70 : DIST(COND:=COND,MD0=>MD850,MD1=>MD851,MD2=>MD852,MD3=>MD853,MD4=>MD854);
71 : DIST(COND:=COND,MD0=>MD855,MD1=>MD856,MD2=>MD857,MD3=>MD858,MD4=>MD859);
72 : DIST(COND:=COND,MD0=>MD860,MD1=>MD861,MD2=>MD862,MD3=>MD863,MD4=>MD864);
73 : DIST(COND:=COND,MD0=>MD865,MD1=>MD866,MD2=>MD867,MD3=>MD868,MD4=>MD869);
74 : DIST(COND:=COND,MD0=>MD870,MD1=>MD871,MD2=>MD872,MD3=>MD873,MD4=>MD874);
75 : DIST(COND:=COND,MD0=>MD875,MD1=>MD876,MD2=>MD877,MD3=>MD878,MD4=>MD879);
76 : DIST(COND:=COND,MD0=>MD880,MD1=>MD881,MD2=>MD882,MD3=>MD883,MD4=>MD884);
77 : DIST(COND:=COND,MD0=>MD885,MD1=>MD886,MD2=>MD887,MD3=>MD888,MD4=>MD889);
78 : DIST(COND:=COND,MD0=>MD890,MD1=>MD891,MD2=>MD892,MD3=>MD893,MD4=>MD894);
79 : DIST(COND:=COND,MD0=>MD895,MD1=>MD896,MD2=>MD897,MD3=>MD898,MD4=>MD899);

80 : DIST(COND:=COND,MD0=>MD900,MD1=>MD901,MD2=>MD902,MD3=>MD903,MD4=>MD904);
81 : DIST(COND:=COND,MD0=>MD905,MD1=>MD906,MD2=>MD907,MD3=>MD908,MD4=>MD909);
82 : DIST(COND:=COND,MD0=>MD910,MD1=>MD911,MD2=>MD912,MD3=>MD913,MD4=>MD914);
83 : DIST(COND:=COND,MD0=>MD915,MD1=>MD916,MD2=>MD917,MD3=>MD918,MD4=>MD919);
84 : DIST(COND:=COND,MD0=>MD920,MD1=>MD921,MD2=>MD922,MD3=>MD923,MD4=>MD924);
85 : DIST(COND:=COND,MD0=>MD925,MD1=>MD926,MD2=>MD927,MD3=>MD928,MD4=>MD929);
86 : DIST(COND:=COND,MD0=>MD930,MD1=>MD931,MD2=>MD932,MD3=>MD933,MD4=>MD934);
87 : DIST(COND:=COND,MD0=>MD935,MD1=>MD936,MD2=>MD937,MD3=>MD938,MD4=>MD939);
88 : DIST(COND:=COND,MD0=>MD940,MD1=>MD941,MD2=>MD942,MD3=>MD943,MD4=>MD944);
89 : DIST(COND:=COND,MD0=>MD945,MD1=>MD946,MD2=>MD947,MD3=>MD948,MD4=>MD949);

90 : DIST(COND:=COND,MD0=>MD950,MD1=>MD951,MD2=>MD952,MD3=>MD953,MD4=>MD954);
91 : DIST(COND:=COND,MD0=>MD955,MD1=>MD956,MD2=>MD957,MD3=>MD958,MD4=>MD959);
92 : DIST(COND:=COND,MD0=>MD960,MD1=>MD961,MD2=>MD962,MD3=>MD963,MD4=>MD964);
93 : DIST(COND:=COND,MD0=>MD965,MD1=>MD966,MD2=>MD967,MD3=>MD968,MD4=>MD969);
94 : DIST(COND:=COND,MD0=>MD970,MD1=>MD971,MD2=>MD972,MD3=>MD973,MD4=>MD974);
95 : DIST(COND:=COND,MD0=>MD975,MD1=>MD976,MD2=>MD977,MD3=>MD978,MD4=>MD979);
96 : DIST(COND:=COND,MD0=>MD980,MD1=>MD981,MD2=>MD982,MD3=>MD983,MD4=>MD984);
97 : DIST(COND:=COND,MD0=>MD985,MD1=>MD986,MD2=>MD987,MD3=>MD988,MD4=>MD989);
98 : DIST(COND:=COND,MD0=>MD990,MD1=>MD991,MD2=>MD992,MD3=>MD993,MD4=>MD994);
99 : DIST(COND:=COND,MD0=>MD995,MD1=>MD996,MD2=>MD997,MD3=>MD998,MD4=>MD999);

END_CASE;
          
END_FUNCTION_BLOCK

(* Запись элемента в выходные массивы *)
FUNCTION_BLOCK WriteItem
  VAR_INPUT
    PIT : TPos8 := -1;  (* Индекс элемента в массиве ITS *)
  END_VAR
  VAR
    Cond : TCond;  (* Состояние элемента *)
    msg : STRING := '';  (* TEST *)
    _SetCond : SetCond;
  END_VAR

            (* Запись состояния в регистры *)
Cond    := get_cn(PIT);
Cond.ID := it_id(PIT);
(*TEST*)
(* #53 - ID = 16761, 0x4179, REG = 3578-3587 *)
(*
if (Cond.ID = 16761) then 
  msg := MakeMsg(msg, '= TEST1 [', ID2Str(IT_ID(PIT)), ',');
  msg := MakeMsg(msg, SINT_TO_STRING(PIT), ',');
  msg := MakeMsg(msg, 'Tmid=', REAL_TO_STRING(INT_TO_REAL(Cond.Tmid)/100.0), ',');
  msg := MakeMsg(msg, 'Tmax=', REAL_TO_STRING(INT_TO_REAL(Cond.Tmax.v)/100.0), ',');
  msg := MakeMsg(msg,  INT_TO_STRING(Cond.Tmax.i[0]), ',');
  msg := MakeMsg(msg,  INT_TO_STRING(Cond.Tmax.i[1]), ',');
  msg := MakeMsg(msg,  INT_TO_STRING(Cond.Tmax.i[2]), ']');
  msg := LogMsg(msg);
end_if;
*)
_SetCond(I := SINT_TO_UINT(PIT), COND := Cond);
          
END_FUNCTION_BLOCK

(* Вывод результатов в регистры *)
PROGRAM P_RES
  VAR_EXTERNAL
    f_Res : BOOL;  (* Флаг выкладки результатов *)
    HDR : THead;  (* Заголовок модели *)
    ITS : TItems;  (* Массив элементов модели *)
  END_VAR
  VAR
    pit : TPos8 := 0;  (* Позиция элемента *)
    Sh : TShape;  (* Фигура элемента *)
    Pt : TPoint;  (* Точка *)
    Off : P_INT;  (* Offset *)
    PGR : TPos8 := -1;  (* Позиция сетки *)
    I : INT := 0;  (* Индекс сетки X *)
    J : INT := 0;  (* Индекс сетки Y *)
    K : INT := 0;  (* Индекс сетки Z *)
    Dot : TDot;  (* Точка сетки *)
    bRes : BOOL := false;  (* Бинарный результат *)
    iRes : TError := E_SUCCESS;  (* Код ошибки *)
    iLog : INT := 0;  (* Счётчик строк протокола *)
    msg : STRING := '';  (* Сообщение в протокол *)
    _WriteItem : WriteItem;  (* Функция записи элемента *)
    _Grid2ul : Grid2ul;
    _GetHead : GetHead;
  END_VAR

            (* Считывание заголовка *)
_GetHead(HEAD => HDR);

(* Test *)
(* if (HDR.ID = 100)  then HDR.ID := 99; end_if; *)
(*
HDR.ID := 100;
HDR.Ax := 2;
HDR.pX := 1800;
HDR.pY := 620;
HDR.pZ := 1575;
*)
(* =1= Протоколирование на консоль === *)
bRes := Do_LogCond(ID2PIT(0));

(* =2= Запись массива элементов в регистры === *)
(*msg:=LogMsg('Write items ... '); *)
FOR pit := 0 TO HDR.Ni-1 DO 
  _WriteItem(PIT := pit);
  (*
  if (len(msg)=0) then msg := MakeMsg(' - Updated items: '); end_if;
  msg := MakeMsg(msg, ' [', ID2Str(IT_ID(pit)), ',');
  msg := MakeMsg(msg,       SINT_TO_STRING(pit), ']');
  if (mod((pit+1),5)=0) then msg:=LogMsg(MakeMsg(msg, ';')); end_if;
  *)
END_FOR; 
(* if (len(msg)>0) then msg:=LogMsg(MakeMsg(msg, ';')); end_if; *)

(* =3= Вывод T-поля объекта [POS=HDR.ID] в регистры === *)
msg:=LogMsg(MakeMsg(msg, '===== T-Field START ====='));      

pit := UINT_TO_SINT(HDR.ID); (* it_pos(ID2PIT(HDR.ID)); *)
if (pit >= 0 and pit < HDR.Ni) then 

  (* Вывод поля обычного элемента *)
  Sh := get_sh(pit);
  _Grid2ul(HGR := its_gr(0), PGR := pit, SH := Sh, iRes=>iRes);
  
elsif (pit = 100) then (* Вывод поля поверхности *)
  
  Sh := _surf(
    ID2PIT(0), 
    UINT_TO_USINT(HDR.Ax), 
    INT_TO_REAL(HDR.pX), 
    INT_TO_REAL(HDR.pY), 
    INT_TO_REAL(HDR.pZ)
  );
  (*Sh := get_sh(0);*)
  ITS.Sh[pit] := Sh;
  
  (* Линковка узлов *)
  iLog := 0;
  for I:=0 to Sh.Kn[0]-1 do
    for J:=0 to Sh.Kn[1]-1 do
      for K:=0 to Sh.Kn[2]-1 do
      
        Dot := link_var(its_gr2(0), 0, Sh, I, J, K);
        (*
        Pt  := Sh_Dot2Point(Sh, I, J, K);
        Dot := Do_FindDot(Pt[0], Pt[1], Pt[2]);
        Off := knoff(Sh.Kn[0], Sh.Kn[1], Sh.Kn[2], I,J,K);
        PGR := set_var( its_gr2(0), 0, Off, _ref(int_to_sint(Dot.v), Dot));
        *)
        
        (*
        if (false or iLog<80) then  
          if (len(msg)=0) then msg := MakeMsg(' =!=> '); end_if;
          msg := MakeMsg(msg, '[', INT_TO_STRING(REAL_TO_INT(Pt[0])), ',');
          msg := MakeMsg(msg,  '', INT_TO_STRING(REAL_TO_INT(Pt[1])), ',');
          msg := MakeMsg(msg,  '', INT_TO_STRING(REAL_TO_INT(Pt[2])), ']');
          if (mod((iLog+1),8)=0) then msg:=LogMsg(MakeMsg(msg, ';')); end_if;
          iLog:=iLog+1;
        end_if;
        *)
        (*
        if (iLog<80) then  
          if (len(msg)=0) then msg := MakeMsg(' =!=> '); end_if;
          msg := MakeMsg(msg, '[', INT_TO_STRING(Dot.v), ',');
          msg := MakeMsg(msg,  '', INT_TO_STRING(Dot.a[0]), ',');
          msg := MakeMsg(msg,  '', INT_TO_STRING(Dot.a[1]), ',');
          msg := MakeMsg(msg,  '', INT_TO_STRING(Dot.a[2]), ']');
          if (mod((iLog+1),8)=0) then msg:=LogMsg(MakeMsg(msg, ';')); end_if;
          iLog:=iLog+1;
        end_if;
        *)
      end_for;
    end_for;
  end_for;
  if (len(msg)>0) then msg:=LogMsg(MakeMsg(msg, ';')); end_if;
  
  _Grid2ul(HGR := its_gr2(0), PGR := 0, SH := Sh, iRes=>iRes);
  
else (* ошибка позиции *)
  {}

end_if;
msg:=LogMsg(MakeMsg(msg, '===== T-Field (END) ====='));      

(* Сброс флага *)
f_Res := FALSE;

          
END_PROGRAM

FUNCTION UDI2REAL : REAL
  VAR_INPUT
    VALUE : UDINT := 0;
  END_VAR
  VAR
    tmp : REAL := 0.0;
  END_VAR

            {{
  union { UDINT  udint; float real; } value;
  value.udint = VALUE;
  TMP = value.real;
}}
UDI2REAL := TMP;

          
END_FUNCTION

(* Компоновка материала *)
FUNCTION m_mat : TMat
  VAR_INPUT
    MD0 : UDINT;
    MD1 : UDINT;
    MD2 : UDINT;
    MD3 : UDINT;
  END_VAR

            m_mat.KT := UDI2REAL(MD0);
m_mat.CP := UDI2REAL(MD1);
m_mat.PL := UDI2REAL(MD2);
m_mat.MD := UDI2REAL(MD3);

          
END_FUNCTION

(* Чтение материала из регистров *)
FUNCTION_BLOCK GetMat
  VAR_EXTERNAL
    MD22 : UDINT;
    MD23 : UDINT;
    MD24 : UDINT;
    MD25 : UDINT;
    MD26 : UDINT;
    MD27 : UDINT;
    MD28 : UDINT;
    MD29 : UDINT;
    MD30 : UDINT;
    MD31 : UDINT;
    MD32 : UDINT;
    MD33 : UDINT;
    MD34 : UDINT;
    MD35 : UDINT;
    MD36 : UDINT;
    MD37 : UDINT;
    MD38 : UDINT;
    MD39 : UDINT;
    MD40 : UDINT;
    MD41 : UDINT;
    MD42 : UDINT;
    MD43 : UDINT;
    MD44 : UDINT;
    MD45 : UDINT;
    MD46 : UDINT;
    MD47 : UDINT;
    MD48 : UDINT;
    MD49 : UDINT;
    MD50 : UDINT;
    MD51 : UDINT;
    MD52 : UDINT;
    MD53 : UDINT;
    MD54 : UDINT;
    MD55 : UDINT;
    MD56 : UDINT;
    MD57 : UDINT;
    MD58 : UDINT;
    MD59 : UDINT;
    MD60 : UDINT;
    MD61 : UDINT;
    MD62 : UDINT;
    MD63 : UDINT;
    MD64 : UDINT;
    MD65 : UDINT;
    MD66 : UDINT;
    MD67 : UDINT;
    MD68 : UDINT;
    MD69 : UDINT;
  END_VAR
  VAR_INPUT
    I : SINT := 0;  (* Индекс материала *)
  END_VAR
  VAR_OUTPUT
    MAT : TMat;  (* Объект "материал" *)
  END_VAR

            CASE i OF
0 : MAT := m_mat(MD22,MD23,MD24,MD25);
1 : MAT := m_mat(MD26,MD27,MD28,MD29);
2 : MAT := m_mat(MD30,MD31,MD32,MD33);
3 : MAT := m_mat(MD34,MD35,MD36,MD37);
4 : MAT := m_mat(MD38,MD39,MD40,MD41);
5 : MAT := m_mat(MD42,MD43,MD44,MD45);
6 : MAT := m_mat(MD46,MD47,MD48,MD49);
7 : MAT := m_mat(MD50,MD51,MD52,MD53);
8 : MAT := m_mat(MD54,MD55,MD56,MD57);
9 : MAT := m_mat(MD58,MD59,MD60,MD61);
10: MAT := m_mat(MD62,MD63,MD64,MD65);
11: MAT := m_mat(MD66,MD67,MD68,MD69);
END_CASE;
          
END_FUNCTION_BLOCK

(* Компоновка профиля *)
FUNCTION m_prof : TProf
  VAR_INPUT
    MD0 : UDINT;
    MD1 : UDINT;
    MD2 : UDINT;
    MD3 : UDINT;
    MD4 : UDINT;
    MD5 : UDINT;
  END_VAR

            m_prof[0].A := UINT_TO_SINT(UDINT_TO_UINT(MD0/65536)/256);
m_prof[0].B := UINT_TO_SINT(mod(UDINT_TO_UINT(MD0/65536),256));
m_prof[1].A := UINT_TO_SINT(UDINT_TO_UINT(mod(MD0,65536))/256);
m_prof[1].B := UINT_TO_SINT(mod(UDINT_TO_UINT(mod(MD0,65536)),256));

m_prof[2].A := UINT_TO_SINT(UDINT_TO_UINT(MD1/65536)/256);
m_prof[2].B := UINT_TO_SINT(mod(UDINT_TO_UINT(MD1/65536),256));
m_prof[3].A := UINT_TO_SINT(UDINT_TO_UINT(mod(MD1,65536))/256);
m_prof[3].B := UINT_TO_SINT(mod(UDINT_TO_UINT(mod(MD1,65536)),256));

m_prof[4].A := UINT_TO_SINT(UDINT_TO_UINT(MD2/65536)/256);
m_prof[4].B := UINT_TO_SINT(mod(UDINT_TO_UINT(MD2/65536),256));
m_prof[5].A := UINT_TO_SINT(UDINT_TO_UINT(mod(MD2,65536))/256);
m_prof[5].B := UINT_TO_SINT(mod(UDINT_TO_UINT(mod(MD2,65536)),256));

m_prof[6].A := UINT_TO_SINT(UDINT_TO_UINT(MD3/65536)/256);
m_prof[6].B := UINT_TO_SINT(mod(UDINT_TO_UINT(MD3/65536),256));
m_prof[7].A := UINT_TO_SINT(UDINT_TO_UINT(mod(MD3,65536))/256);
m_prof[7].B := UINT_TO_SINT(mod(UDINT_TO_UINT(mod(MD3,65536)),256));

m_prof[8].A := UINT_TO_SINT(UDINT_TO_UINT(MD4/65536)/256);
m_prof[8].B := UINT_TO_SINT(mod(UDINT_TO_UINT(MD4/65536),256));
m_prof[9].A := UINT_TO_SINT(UDINT_TO_UINT(mod(MD4,65536))/256);
m_prof[9].B := UINT_TO_SINT(mod(UDINT_TO_UINT(mod(MD4,65536)),256));

m_prof[10].A := UINT_TO_SINT(UDINT_TO_UINT(MD5/65536)/256);
m_prof[10].B := UINT_TO_SINT(mod(UDINT_TO_UINT(MD5/65536),256));
m_prof[11].A := UINT_TO_SINT(UDINT_TO_UINT(mod(MD5,65536))/256);
m_prof[11].B := UINT_TO_SINT(mod(UDINT_TO_UINT(mod(MD5,65536)),256));

          
END_FUNCTION

(* Чтение профиля из регистров *)
FUNCTION_BLOCK GetProf
  VAR_EXTERNAL
    MD120 : UDINT;
    MD121 : UDINT;
    MD122 : UDINT;
    MD123 : UDINT;
    MD124 : UDINT;
    MD125 : UDINT;
    MD126 : UDINT;
    MD127 : UDINT;
    MD128 : UDINT;
    MD129 : UDINT;
    MD130 : UDINT;
    MD131 : UDINT;
    MD132 : UDINT;
    MD133 : UDINT;
    MD134 : UDINT;
    MD135 : UDINT;
    MD136 : UDINT;
    MD137 : UDINT;
    MD138 : UDINT;
    MD139 : UDINT;
    MD140 : UDINT;
    MD141 : UDINT;
    MD142 : UDINT;
    MD143 : UDINT;
    MD144 : UDINT;
    MD145 : UDINT;
    MD146 : UDINT;
    MD147 : UDINT;
    MD148 : UDINT;
    MD149 : UDINT;
    MD150 : UDINT;
    MD151 : UDINT;
    MD152 : UDINT;
    MD153 : UDINT;
    MD154 : UDINT;
    MD155 : UDINT;
    MD156 : UDINT;
    MD157 : UDINT;
    MD158 : UDINT;
    MD159 : UDINT;
    MD160 : UDINT;
    MD161 : UDINT;
    MD162 : UDINT;
    MD163 : UDINT;
    MD164 : UDINT;
    MD165 : UDINT;
    MD166 : UDINT;
    MD167 : UDINT;
    MD168 : UDINT;
    MD169 : UDINT;
    MD170 : UDINT;
    MD171 : UDINT;
    MD172 : UDINT;
    MD173 : UDINT;
    MD174 : UDINT;
    MD175 : UDINT;
    MD176 : UDINT;
    MD177 : UDINT;
    MD178 : UDINT;
    MD179 : UDINT;
    MD180 : UDINT;
    MD181 : UDINT;
    MD182 : UDINT;
    MD183 : UDINT;
    MD184 : UDINT;
    MD185 : UDINT;
    MD186 : UDINT;
    MD187 : UDINT;
    MD188 : UDINT;
    MD189 : UDINT;
    MD190 : UDINT;
    MD191 : UDINT;
    MD192 : UDINT;
    MD193 : UDINT;
    MD194 : UDINT;
    MD195 : UDINT;
    MD196 : UDINT;
    MD197 : UDINT;
    MD198 : UDINT;
    MD199 : UDINT;
    MD200 : UDINT;
    MD201 : UDINT;
    MD202 : UDINT;
    MD203 : UDINT;
    MD204 : UDINT;
    MD205 : UDINT;
    MD206 : UDINT;
    MD207 : UDINT;
    MD208 : UDINT;
    MD209 : UDINT;
    MD210 : UDINT;
    MD211 : UDINT;
    MD212 : UDINT;
    MD213 : UDINT;
    MD214 : UDINT;
    MD215 : UDINT;
    MD216 : UDINT;
    MD217 : UDINT;
    MD218 : UDINT;
    MD219 : UDINT;
    MD220 : UDINT;
    MD221 : UDINT;
    MD222 : UDINT;
    MD223 : UDINT;
    MD224 : UDINT;
    MD225 : UDINT;
    MD226 : UDINT;
    MD227 : UDINT;
    MD228 : UDINT;
    MD229 : UDINT;
    MD230 : UDINT;
    MD231 : UDINT;
    MD232 : UDINT;
    MD233 : UDINT;
    MD234 : UDINT;
    MD235 : UDINT;
    MD236 : UDINT;
    MD237 : UDINT;
    MD238 : UDINT;
    MD239 : UDINT;
    MD240 : UDINT;
    MD241 : UDINT;
    MD242 : UDINT;
    MD243 : UDINT;
    MD244 : UDINT;
    MD245 : UDINT;
    MD246 : UDINT;
    MD247 : UDINT;
    MD248 : UDINT;
    MD249 : UDINT;
    MD250 : UDINT;
    MD251 : UDINT;
    MD252 : UDINT;
    MD253 : UDINT;
    MD254 : UDINT;
    MD255 : UDINT;
    MD256 : UDINT;
    MD257 : UDINT;
    MD258 : UDINT;
    MD259 : UDINT;
    MD260 : UDINT;
    MD261 : UDINT;
    MD262 : UDINT;
    MD263 : UDINT;
    MD264 : UDINT;
    MD265 : UDINT;
    MD266 : UDINT;
    MD267 : UDINT;
    MD268 : UDINT;
    MD269 : UDINT;
    MD270 : UDINT;
    MD271 : UDINT;
    MD272 : UDINT;
    MD273 : UDINT;
    MD274 : UDINT;
    MD275 : UDINT;
    MD276 : UDINT;
    MD277 : UDINT;
    MD278 : UDINT;
    MD279 : UDINT;
    MD280 : UDINT;
    MD281 : UDINT;
    MD282 : UDINT;
    MD283 : UDINT;
    MD284 : UDINT;
    MD285 : UDINT;
    MD286 : UDINT;
    MD287 : UDINT;
    MD288 : UDINT;
    MD289 : UDINT;
    MD290 : UDINT;
    MD291 : UDINT;
    MD292 : UDINT;
    MD293 : UDINT;
    MD294 : UDINT;
    MD295 : UDINT;
    MD296 : UDINT;
    MD297 : UDINT;
    MD298 : UDINT;
    MD299 : UDINT;
  END_VAR
  VAR_INPUT
    I : SINT := 0;  (* Индекс профиля *)
  END_VAR
  VAR_OUTPUT
    PROF : TProf;  (* Объект "профиль" *)
  END_VAR

            CASE i OF
0 : PROF := m_prof(MD120,MD121,MD122,MD123,MD124,MD125);
1 : PROF := m_prof(MD126,MD127,MD128,MD129,MD130,MD131);
2 : PROF := m_prof(MD132,MD133,MD134,MD135,MD136,MD137);
3 : PROF := m_prof(MD138,MD139,MD140,MD141,MD142,MD143);
4 : PROF := m_prof(MD144,MD145,MD146,MD147,MD148,MD149);
5 : PROF := m_prof(MD150,MD151,MD152,MD153,MD154,MD155);
6 : PROF := m_prof(MD156,MD157,MD158,MD159,MD160,MD161);
7 : PROF := m_prof(MD162,MD163,MD164,MD165,MD166,MD167);
8 : PROF := m_prof(MD168,MD169,MD170,MD171,MD172,MD173);
9 : PROF := m_prof(MD174,MD175,MD176,MD177,MD178,MD179);
10: PROF := m_prof(MD180,MD181,MD182,MD183,MD184,MD185);
11: PROF := m_prof(MD186,MD187,MD188,MD189,MD190,MD191);
12: PROF := m_prof(MD192,MD193,MD194,MD195,MD196,MD197);
13: PROF := m_prof(MD198,MD199,MD200,MD201,MD202,MD203);
14: PROF := m_prof(MD204,MD205,MD206,MD207,MD208,MD209);
15: PROF := m_prof(MD210,MD211,MD212,MD213,MD214,MD215);
16: PROF := m_prof(MD216,MD217,MD218,MD219,MD220,MD221);
17: PROF := m_prof(MD222,MD223,MD224,MD225,MD226,MD227);
18: PROF := m_prof(MD228,MD229,MD230,MD231,MD232,MD233);
19: PROF := m_prof(MD234,MD235,MD236,MD237,MD238,MD239);
20: PROF := m_prof(MD240,MD241,MD242,MD243,MD244,MD245);
21: PROF := m_prof(MD246,MD247,MD248,MD249,MD250,MD251);
22: PROF := m_prof(MD252,MD253,MD254,MD255,MD256,MD257);
23: PROF := m_prof(MD258,MD259,MD260,MD261,MD262,MD263);
24: PROF := m_prof(MD264,MD265,MD266,MD267,MD268,MD269);
25: PROF := m_prof(MD270,MD271,MD272,MD273,MD274,MD275);
26: PROF := m_prof(MD276,MD277,MD278,MD279,MD280,MD281);
27: PROF := m_prof(MD282,MD283,MD284,MD285,MD286,MD287);
28: PROF := m_prof(MD288,MD289,MD290,MD291,MD292,MD293);
29: PROF := m_prof(MD294,MD295,MD296,MD297,MD298,MD299);
END_CASE;
          
END_FUNCTION_BLOCK

(* Компоновка величины *)
FUNCTION m_val : TVal
  VAR_INPUT
    MD0 : UDINT;
    MD1 : UDINT;
  END_VAR

            m_val.Iv      := UDINT_TO_INT(MD0/65536);
m_val.Vi[0].A := UINT_TO_SINT(UDINT_TO_UINT(mod(MD0,65536))/256);
m_val.Vi[0].B := UINT_TO_SINT(mod(UDINT_TO_UINT(mod(MD0,65536)),256));
m_val.Vi[1].A := UINT_TO_SINT(UDINT_TO_UINT(MD1/65536)/256);
m_val.Vi[1].B := UINT_TO_SINT(mod(UDINT_TO_UINT(MD1/65536),256));
m_val.Vi[2].A := UINT_TO_SINT(UDINT_TO_UINT(mod(MD1,65536))/256);
m_val.Vi[2].B := UINT_TO_SINT(mod(UDINT_TO_UINT(mod(MD1,65536)),256));



          
END_FUNCTION

(* Чтение величины из регистров *)
FUNCTION_BLOCK GetVal
  VAR_EXTERNAL
    MD70 : UDINT;
    MD71 : UDINT;
    MD72 : UDINT;
    MD73 : UDINT;
    MD74 : UDINT;
    MD75 : UDINT;
    MD76 : UDINT;
    MD77 : UDINT;
    MD78 : UDINT;
    MD79 : UDINT;
    MD80 : UDINT;
    MD81 : UDINT;
    MD82 : UDINT;
    MD83 : UDINT;
    MD84 : UDINT;
    MD85 : UDINT;
    MD86 : UDINT;
    MD87 : UDINT;
    MD88 : UDINT;
    MD89 : UDINT;
    MD90 : UDINT;
    MD91 : UDINT;
    MD92 : UDINT;
    MD93 : UDINT;
    MD94 : UDINT;
    MD95 : UDINT;
    MD96 : UDINT;
    MD97 : UDINT;
    MD98 : UDINT;
    MD99 : UDINT;
    MD100 : UDINT;
    MD101 : UDINT;
    MD102 : UDINT;
    MD103 : UDINT;
    MD104 : UDINT;
    MD105 : UDINT;
    MD106 : UDINT;
    MD107 : UDINT;
    MD108 : UDINT;
    MD109 : UDINT;
    MD110 : UDINT;
    MD111 : UDINT;
    MD112 : UDINT;
    MD113 : UDINT;
    MD114 : UDINT;
    MD115 : UDINT;
    MD116 : UDINT;
    MD117 : UDINT;
    MD118 : UDINT;
    MD119 : UDINT;
  END_VAR
  VAR_INPUT
    I : SINT := 0;  (* Индекс величины *)
  END_VAR
  VAR_OUTPUT
    VAL : TVal;  (* Объект "величина" *)
  END_VAR

            CASE i OF
0 : VAL := m_val(MD70,MD71);
1 : VAL := m_val(MD72,MD73);
2 : VAL := m_val(MD74,MD75);
3 : VAL := m_val(MD76,MD77);
4 : VAL := m_val(MD78,MD79);
5 : VAL := m_val(MD80,MD81);
6 : VAL := m_val(MD82,MD83);
7 : VAL := m_val(MD84,MD85);
8 : VAL := m_val(MD86,MD87);
9 : VAL := m_val(MD88,MD89);
10: VAL := m_val(MD90,MD91);
11: VAL := m_val(MD92,MD93);
12: VAL := m_val(MD94,MD95);
13: VAL := m_val(MD96,MD97);
14: VAL := m_val(MD98,MD99);
15: VAL := m_val(MD100,MD101);
16: VAL := m_val(MD102,MD103);
17: VAL := m_val(MD104,MD105);
18: VAL := m_val(MD106,MD107);
19: VAL := m_val(MD108,MD109);
20: VAL := m_val(MD110,MD111);
21: VAL := m_val(MD112,MD113);
22: VAL := m_val(MD114,MD115);
23: VAL := m_val(MD116,MD117);
24: VAL := m_val(MD118,MD119);
END_CASE;
          
END_FUNCTION_BLOCK

(* Алгоритм "Быстрая сортировка" *)
FUNCTION_BLOCK Sort_IDS
  VAR_EXTERNAL
    ITS : TItems;  (* Массив элементов *)
  END_VAR
  VAR_INPUT
    iBegin : TPos8 := 0;  (* Индекс начала сортировки *)
    iEnd : TPos8 := 0;  (* Индекс завершения сортировки *)
  END_VAR
  VAR_OUTPUT
    iRes : TError := E_SUCCESS;  (* Результат выполнения *)
  END_VAR
  VAR
    iL : TPos8;  (* Левая граница *)
    iR : TPos8;  (* Правая граница *)
    LL : TPos8;  (* Левый индекс *)
    RR : TPos8;  (* Правый индекс *)
    Z : P_IDPIT;  (* Средний элемент для сравнения *)
    iS : TPos8;  (* Индекс стека *)
    Stack : ARRAY[0..49] OF TPos8;  (* Стек индексов элементов *)
    fBreak : BOOL;  (* Флаг завершения внешнего цикла *)
    tmp : P_IDPIT;  (* Буфер обмена значениями *)
  END_VAR

            (* Начальные значения *)
iRes  := E_SUCCESS;				
iS    := 0; 
iL    := iBegin; 
iR    := iEnd; 

fBreak := false;
WHILE NOT fBreak DO         (* внешний цикл = "рекурсия" *)
  
	IF iL < iR THEN
    (* Значение среднего элемента в качестве опорного значения *)
		Z := ITS.Pr[WORD_TO_SINT(SHR(UINT_TO_WORD(SINT_TO_UINT(iR)+SINT_TO_UINT(iL)),1))]; 
    
		LL := iL; RR := iR;
		WHILE (LL <= RR) DO     (* внутренний цикл = выделение частей *)
 			(* Сравнение - возрастающий порядок *)
      while (ITS.Pr[LL].A < Z.A) do LL:=LL+1; end_while;
      while (ITS.Pr[RR].A > Z.A) do RR:=RR-1; end_while;
			if LL <= RR then  
        if (LL <> RR) then  (* Обмен значений *)
          tmp := ITS.Pr[RR]; 
          ITS.Pr[RR] := ITS.Pr[LL]; 
          ITS.Pr[LL] := tmp; 
        end_if;        
        LL:=LL+1; RR:=RR-1;
			end_if;
		END_WHILE;

		(* Вставка в стек *)
		IF iS < 49 THEN 
      Stack[iS] := iR;		  (* Отложенная сортировка правой части  *)
      iS := iS+1; 
    ELSE                    (* Стек выбран - ошибка величины стека *)
      fBreak := TRUE; 
      iRes := E_STACKSIZE; 
    END_IF;
      
		iR := MAX(iL, LL-1);    (* Сортировка левой части - в следующем цикле *)
    
  ELSE
    
		IF iS > 0 THEN          (* Теперь сортируем правую часть *)
			iL := iR+1;
			(* Выборка из стека *)
			iS := iS-1;	
			iR:= Stack[iS];
		ELSE                    (* Стек выбран - конец работы *)
      fBreak := TRUE;
		END_IF;
    
	END_IF;
  
END_WHILE; (* Сортировка завершена *)

          
END_FUNCTION_BLOCK

(* Чтение конфигурации из регистров *)
PROGRAM P_CONF
  VAR_EXTERNAL
    STAT : TStat;  (* Состояние выполнения *)
    f_Conf : BOOL;  (* Флаг конфигурирования *)
    HDR : THead;  (* Заголовок модели *)
    STS : TSets;  (* Массив конфигураций *)
    ITS : TItems;  (* Массив элементов *)
  END_VAR
  VAR
    msg : STRING;  (* Строка сообщения *)
    _GetHead : GetHead;  (* ФБ чтения заголовка *)
    _GetMat : GetMat;  (* ФБ чтения материалов *)
    _GetVal : GetVal;  (* ФБ чтения связанных величин *)
    _GetProf : GetProf;  (* ФБ чтения профилей *)
    _ReadItem : ReadItem;  (* ФБ чтения элементов *)
    _Sort_IDS : Sort_IDS;  (* ФБ "быстрая сортировка" *)
    _Process_X : Process_XYZ;
  END_VAR

            (* Локальные переменные *)
VAR
  i,j,k,l : SINT;      (* Индексы в массивах              *)
  iLev    : SINT;      (* Уровень элемента                *)
  pit,idx : TPos8;     (* Индексы элементов               *)
  iPar    : TPos8;     (* Индекс родителя                 *)
  iPrev   : TPos8;     (* Индекс предыдущего элемента     *)
  nRes    : TError;    (* Код результата выполнения       *)
  iRes    : INT;       (* Возвращаемое значение           *)
  it      : TITER;     (* Итератор для обхода дерева      *)
  btRes   : BYTE;      (* Результат проверки точки модели *)
  bRes    : BOOL;
  rRes    : REAL;
  ii      : DINT;
  sibt    : P_SIBT;
END_VAR

(* Установка начальных значений *)
{{
  // Инициализация фиктивного элемента
  //TITEM *pItem0 = __GET_GLOBAL_DUMMY();
  //memset(pItem0,0x00,sizeof(TITEM));
  //pItem0->ID = 0xffff;
  
  // Инициализация состояния ресурса
  TSTAT *pStat = __GET_GLOBAL_STAT();
  *pStat = (TSTAT) {FALSE, TRUE, TERROR__E_SUCCESS, 0, __INIT_STRING};
}}

nRes := E_SUCCESS;          (* Установка кода результата    *)
bRes := st_set_debug(TRUE); (* Установка флага отладки      *) 

msg  := LogMsg('== CONFIG ...');

(* === Чтение и валидация заголовка === *)
_GetHead(HEAD => HDR);

msg := MakeMsg(' - Read header ... (');
msg := MakeMsg(msg, SINT_TO_STRING(HDR.Ni), ', ');
msg := MakeMsg(msg, SINT_TO_STRING(HDR.Nm), ', ');
msg := MakeMsg(msg, SINT_TO_STRING(HDR.Nv), ', ');
msg := MakeMsg(msg, SINT_TO_STRING(HDR.Np), ')');

(* Валидация заголовка *)
if (HDR.Ni= 0 or HDR.Ni>100) then nRes:=E_HEAD; {goto __exit} end_if;
if (HDR.Nm= 0 or HDR.Nm>12)  then nRes:=E_HEAD; {goto __exit} end_if;
if (HDR.Nv< 0 or HDR.Nv>25)  then nRes:=E_HEAD; {goto __exit} end_if;
if (HDR.Np< 0 or HDR.Np>30)  then nRes:=E_HEAD; {goto __exit} end_if;
msg:=LogMsg(MakeMsg(msg, ';'));

(* Проверка периодов расчёта элемента *)
if (HDR.TR[0] = T#0s) then HDR.TR[0]:=T#15s; end_if;
if (HDR.TR[1] = T#0s) then HDR.TR[1]:=T#30s; end_if;
if (HDR.TR[2] = T#0s) then HDR.TR[2]:=T#45s; end_if;
if (HDR.TR[3] = T#0s) then HDR.TR[3]:=T#60s; end_if;

(* === Чтение и валидация массива материалов === *)
msg:=LogMsg('Read materials ... ');
FOR i := 0 TO HDR.Nm-1 DO 
  _GetMat(I:=i, MAT => STS.Mt[i]);
  msg := MakeMsg(' - Get material [', SINT_TO_STRING(i), '] ... (');
  msg := MakeMsg(msg, REAL_TO_STRING(STS.Mt[i].KT), ', ');
  msg := MakeMsg(msg, REAL_TO_STRING(STS.Mt[i].CP), ', ');
  msg := MakeMsg(msg, REAL_TO_STRING(STS.Mt[i].PL), ', ');
  msg := MakeMsg(msg, REAL_TO_STRING(STS.Mt[i].MD), ')');
  (* Валидация *)
  if (STS.Mt[i].KT < 1.0E-8) then nRes:=E_MATER; {goto __exit} end_if;
  if (STS.Mt[i].CP < 1.0E-8) then nRes:=E_MATER; {goto __exit} end_if;
  if (STS.Mt[i].PL < 1.0E-8) then nRes:=E_MATER; {goto __exit} end_if;
  msg:=LogMsg(MakeMsg(msg, ';'));
END_FOR;

(* === Чтение и валидация профилей === *)
msg:=LogMsg('Read profiles ... ');
FOR i := 0 TO HDR.Np-1 DO 
  _GetProf(I:=i, PROF => STS.Pr[i]);
  msg := MakeMsg(' - Get profile [', SINT_TO_STRING(i), '] ...');
  FOR j := 0 TO 11 DO
    msg := MakeMsg(msg, ' (', SINT_TO_STRING(STS.Pr[i][j].A), ',');
    msg := MakeMsg(msg,       SINT_TO_STRING(STS.Pr[i][j].B), ')');
    (* Валидация *)
    if (STS.Pr[i][j].A <    0 or STS.Pr[i][j].A > 100) then nRes:=E_PROFILE; {goto __exit} end_if;
    if (STS.Pr[i][j].B < -100 or STS.Pr[i][j].B > 100) then nRes:=E_PROFILE; {goto __exit} end_if;
  END_FOR;
  msg:=LogMsg(MakeMsg(msg, ';'));
END_FOR;

(* === Чтение и валидация связанных величин === *)
msg:=LogMsg('Read values ... ');
FOR i := 0 TO HDR.Nv-1 DO 
  _GetVal(I:=i, VAL => STS.Vl[i]);
  msg := MakeMsg(' - Get value [', SINT_TO_STRING(i), '] ...');
  if (STS.Vl[i].Iv >=USINT_TO_INT(30) and STS.Vl[i].Iv <> -1) then nRes:=E_VALUE; {goto __exit} end_if;
  FOR j := 0 TO 2 DO
    msg := MakeMsg(msg, ' (', SINT_TO_STRING(STS.Vl[i].Vi[j].A), ',');
    msg := MakeMsg(msg,       SINT_TO_STRING(STS.Vl[i].Vi[j].B), ')');
    (* Валидация *)
    if (STS.Vl[i].Vi[j].A < 0 or STS.Vl[i].Vi[j].A >     100) then nRes:=E_VALUE; {goto __exit} end_if;
    if (STS.Vl[i].Vi[j].B < 0 or STS.Vl[i].Vi[j].B >= HDR.Np) then nRes:=E_VALUE; {goto __exit} end_if;
  END_FOR;
  msg:=LogMsg(MakeMsg(msg, ';'));
END_FOR;

(* === Чтение массива элементов === *)
msg:=LogMsg('Read items ... '); 
FOR pit := 0 TO HDR.Ni-1 DO 
  _ReadItem(PIT := pit, iRes => nRes); 
  
  (* Протоколирование *)
  if (len(msg)=0) then msg := MakeMsg(' - Updated items: '); end_if;
  msg := MakeMsg(msg, ' [', ID2Str(IT_ID(pit)), ',');
  msg := MakeMsg(msg,       SINT_TO_STRING(pit), ']');
  if (mod((pit+1),5)=0) then msg:=LogMsg(MakeMsg(msg, ';')); end_if;
  if (nRes <> E_SUCCESS) then {goto __exit} end_if;
  
  (* Регистрация элемента в массиве IDs (UI->SI)*)
  ITS.Pr[pit].A := ITS.It[pit].ID; 
  ITS.Pr[pit].B := (pit);
END_FOR; 
if (len(msg)>0) then msg:=LogMsg(MakeMsg(msg, ';')); end_if;

(* === Упорядочивание массива по IDs === *)
msg:=LogMsg(MakeMsg('Sort items ... '));
_Sort_IDS(iBegin:=0, iEnd:=HDR.Ni-1, iRes => nRes); 
if (nRes <> E_SUCCESS) then {goto __exit} end_if;

(* === Формирование иерархической структуры === *)
if (ITS.Pr[0].A<>0) then 
  nRes  := E_ROOT; 
  {goto __exit} 
end_if;

(* ROOT settings *)
iPrev := ITS.Pr[0].B;   
iPar  := iPrev;
iLev  := -1;
ITS.It[iPar].Par := -1; 

(* Построение дерева *)
FOR idx := 1 TO HDR.Ni-1 DO
  pit := ITS.Pr[idx].B;   (* Индекс элемента  *)
  l := IT_Lev(pit);       (* Уровень элемента *)
  if (l < 0) then nRes:=E_STRUCT; {goto __exit} end_if;

  (* Определяем индекс родителя iPar *)  
  if (l <> iLev) then     (* Смена уровня вложенности - смена родителя *)
    (* Нахождение родителя для текущего элемента *)
    if (l > iLev) then    (* Спускаемся на уровень вниз  *)
      (* Возможен спуск только на одну ступень (!) *)
      if (l-iLev <> 1) then nRes:=E_STRUCT; {goto __exit} end_if;
      (* Предыдущий элемент должен быть родительским *)
      (*if (not ITS.IT[iPrev].bP) then nRes:=E_STRUCT; {goto __exit} end_if;*)
      iPar := iPrev;      (* Родитель - предыдущий элемент *)
    else                  (* Поднимаемся вверх *)
      (* Вычисление родителя по ступенькам вверх от предыдущего *)
      iPar := iPrev;
      for k := l to iLev do 
        if (iPar<>-1) then iPar := ITS.IT[iPar].Par; end_if;
      end_for;
    end_if;
  else (* Тот же уровень вложенности - родитель не меняется *)
    iPar := iPar;
  end_if;
  (* Родительский элемент должен существовать (!) *)
  if (iPar=-1) then nRes:=E_STRUCT; {goto __exit} end_if;
  
  ITS.It[pit].Par := iPar;      (* Сохраняем индекс родителя              *)
  k := ITS.It[iPar].Num;        (* Читается количество детей              *)
  ITS.It[iPar].Kids[k] := pit;  (* Сохраняем элемент в массиве детей      *)
  ITS.It[iPar].Num := k+1;      (* Увеличиваем счётчик детей              *) 
  iLev  := l;                   (* сохраняем уровень предыдущего элемента *)
  iPrev := pit;                 (* сохраняем индекс  предыдущего элемента *)
END_FOR;

(* === Валидация (подготовка модели) === *)
bRes:=Do_Validate(ID2PIT(0));
msg:=LogMsg(MakeMsg('Validate model ... ', BOOL_TO_STRING(bRes)));
msg:=LogMsg(STAT.STR);

(* === Проверка согласованности модели === *)
bRes:=Do_CheckValid(ID2PIT(0));
msg:=LogMsg(MakeMsg('Model CheckValid ... ', BOOL_TO_STRING(bRes)));
msg:=LogMsg(MakeMsg(STAT.STR));

(* === Линкование элементов === *)
msg:=LogMsg('Model LinkItems ... ');
iRes:=Do_LinkItems(ID2PIT(0));

if (iRes<>-1) then
  msg:=LogMsg(MakeMsg('Model LinkItems ... OK [items -> Air = ', INT_TO_STRING(iRes), '];'));
else
  msg:=LogMsg('Model LinkItems ... FAILED');
end_if;

bRes := st_set_ready(TRUE); (* Установка флага деблокировки *) 

{__exit:}
(* === Протоколирование результата === *)
if (nRes <> E_SUCCESS) then msg:=LogMsg(msg); end_if;
msg:=LogMsg(MakeMsg('== CONFIG -> ', Err2Str(nRes)), Debug, nRes);

f_Conf := FALSE;            (* Сброс флага конфигурирования *)

          
END_PROGRAM

(* 32xUDINT в массив 32xREAL *)
FUNCTION_BLOCK Buffer32
  VAR_INPUT
    MD0 : UDINT;  (* Входной параметр *)
    MD1 : UDINT;  (* Входной параметр *)
    MD2 : UDINT;  (* Входной параметр *)
    MD3 : UDINT;  (* Входной параметр *)
    MD4 : UDINT;  (* Входной параметр *)
    MD5 : UDINT;  (* Входной параметр *)
    MD6 : UDINT;  (* Входной параметр *)
    MD7 : UDINT;  (* Входной параметр *)
    MD8 : UDINT;  (* Входной параметр *)
    MD9 : UDINT;  (* Входной параметр *)
    MD10 : UDINT;  (* Входной параметр *)
    MD11 : UDINT;  (* Входной параметр *)
    MD12 : UDINT;  (* Входной параметр *)
    MD13 : UDINT;  (* Входной параметр *)
    MD14 : UDINT;  (* Входной параметр *)
    MD15 : UDINT;  (* Входной параметр *)
    MD16 : UDINT;  (* Входной параметр *)
    MD17 : UDINT;  (* Входной параметр *)
    MD18 : UDINT;  (* Входной параметр *)
    MD19 : UDINT;  (* Входной параметр *)
    MD20 : UDINT;  (* Входной параметр *)
    MD21 : UDINT;  (* Входной параметр *)
    MD22 : UDINT;  (* Входной параметр *)
    MD23 : UDINT;  (* Входной параметр *)
    MD24 : UDINT;  (* Входной параметр *)
    MD25 : UDINT;  (* Входной параметр *)
    MD26 : UDINT;  (* Входной параметр *)
    MD27 : UDINT;  (* Входной параметр *)
    MD28 : UDINT;  (* Входной параметр *)
    MD29 : UDINT;  (* Входной параметр *)
    MD30 : UDINT;  (* Входной параметр *)
    MD31 : UDINT;  (* Входной параметр *)
  END_VAR
  VAR_OUTPUT
    BUF : ARRAY[0..31] OF REAL;  (* Выходной массив *)
  END_VAR

            BUF[0] :=UDI2REAL(MD0);
BUF[1] :=UDI2REAL(MD1);
BUF[2] :=UDI2REAL(MD2);
BUF[3] :=UDI2REAL(MD3);
BUF[4] :=UDI2REAL(MD4);
BUF[5] :=UDI2REAL(MD5);
BUF[6] :=UDI2REAL(MD6);
BUF[7] :=UDI2REAL(MD7);
BUF[8] :=UDI2REAL(MD8);
BUF[9] :=UDI2REAL(MD9);
BUF[10]:=UDI2REAL(MD10);
BUF[11]:=UDI2REAL(MD11);
BUF[12]:=UDI2REAL(MD12);
BUF[13]:=UDI2REAL(MD13);
BUF[14]:=UDI2REAL(MD14);
BUF[15]:=UDI2REAL(MD15);
BUF[16]:=UDI2REAL(MD16);
BUF[17]:=UDI2REAL(MD17);
BUF[18]:=UDI2REAL(MD18);
BUF[19]:=UDI2REAL(MD19);
BUF[20]:=UDI2REAL(MD20);
BUF[21]:=UDI2REAL(MD21);
BUF[22]:=UDI2REAL(MD22);
BUF[23]:=UDI2REAL(MD23);
BUF[24]:=UDI2REAL(MD24);
BUF[25]:=UDI2REAL(MD25);
BUF[26]:=UDI2REAL(MD26);
BUF[27]:=UDI2REAL(MD27);
BUF[28]:=UDI2REAL(MD28);
BUF[29]:=UDI2REAL(MD29);
BUF[30]:=UDI2REAL(MD30);
BUF[31]:=UDI2REAL(MD31);

          
END_FUNCTION_BLOCK

(* Выкладка заголовка расчёта *)
FUNCTION_BLOCK DistRes
  VAR_OUTPUT
    MD0 : UDINT;
    MD1 : UDINT;
    MD2 : UDINT;
    MD3 : UDINT;
    MD4 : UDINT;
    MD5 : UDINT;
    MD6 : UDINT;
    MD7 : UDINT;
    MD8 : UDINT;
    MD9 : UDINT;
  END_VAR
  VAR_INPUT
    RES : TRes;  (* Объект "Заголовок расчёта модели" *)
  END_VAR

            MD0 := RES.DR;  (* секунд от 01-01-1970 *)
MD1 := TIME_TO_UDINT(RES.TR);
MD2 := TIME_TO_UDINT(RES.FP);
MD3 := UINT_TO_UDINT(RES.ER)*65536 + WORD_TO_UDINT(RES.FL);
MD4 := RES.RV[0];
MD5 := RES.RV[1];
MD6 := RES.RV[2];
MD7 := RES.RV[3];
MD8 := RES.RV[4];
MD9 := RES.RV[5];


          
END_FUNCTION_BLOCK

(* Выкладка фазных параметров *)
FUNCTION_BLOCK DistPhaseO
  VAR_OUTPUT
    MD0 : UDINT;
    MD1 : UDINT;
    MD2 : UDINT;
    MD3 : UDINT;
    MD4 : UDINT;
    MD5 : UDINT;
    MD6 : UDINT;
    MD7 : UDINT;
  END_VAR
  VAR_INPUT
    PhaseO : TPhaseO;  (* Объект "выходные параметры фазы" *)
  END_VAR

            MD0 := REAL_TO_UDINT(PhaseO.Q0);
MD1 := REAL_TO_UDINT(PhaseO.Q1);  
MD2 := REAL_TO_UDINT(PhaseO.Q2);
MD3 := REAL_TO_UDINT(PhaseO.Tin); 
MD4 := REAL_TO_UDINT(PhaseO.Tout);
MD5 := REAL_TO_UDINT(PhaseO.Qm);
MD6 := REAL_TO_UDINT(PhaseO.Se);  
MD7 := REAL_TO_UDINT(PhaseO.Ve);

          
END_FUNCTION_BLOCK

(* Выкладка выходных параметров *)
FUNCTION_BLOCK DistVarO
  VAR_OUTPUT
    MD0 : UDINT;
    MD1 : UDINT;
    MD2 : UDINT;
    MD3 : UDINT;
    MD4 : UDINT;
    MD5 : UDINT;
  END_VAR
  VAR_INPUT
    VarO : TVarO;  (* Объект "выходные параметры" *)
  END_VAR

            MD0 := VarO.DTO;  (* секунд от 01-01-1970 *)
MD1 := TIME_TO_UDINT(VarO.TMO);
MD2 := REAL_TO_UDINT(VarO.QTY);
MD3 := REAL_TO_UDINT(VarO.QTS);
MD4 := REAL_TO_UDINT(VarO.RO1);
MD5 := REAL_TO_UDINT(VarO.RO2);

          
END_FUNCTION_BLOCK

(* Запись заголовка результата *)
FUNCTION_BLOCK SetRes
  VAR_EXTERNAL
    MD490 : UDINT;
    MD491 : UDINT;
    MD492 : UDINT;
    MD493 : UDINT;
    MD494 : UDINT;
    MD495 : UDINT;
    MD496 : UDINT;
    MD497 : UDINT;
    MD498 : UDINT;
    MD499 : UDINT;
  END_VAR
  VAR_INPUT
    RES : TRes;  (* Объект "заголовок результата" *)
  END_VAR
  VAR
    DIST : DistRes;
  END_VAR

            DIST(RES:=RES,MD0=>MD490,MD1=>MD491,MD2=>MD492,MD3=>MD493,MD4=>MD494,
              MD5=>MD495,MD6=>MD496,MD7=>MD497,MD8=>MD498,MD9=>MD499);

          
END_FUNCTION_BLOCK

(* Запись Вых. фазы *)
FUNCTION_BLOCK SetPhaseO
  VAR_EXTERNAL
    MD466 : UDINT;
    MD467 : UDINT;
    MD468 : UDINT;
    MD469 : UDINT;
    MD470 : UDINT;
    MD471 : UDINT;
    MD472 : UDINT;
    MD473 : UDINT;
    MD474 : UDINT;
    MD475 : UDINT;
    MD476 : UDINT;
    MD477 : UDINT;
    MD478 : UDINT;
    MD479 : UDINT;
    MD480 : UDINT;
    MD481 : UDINT;
    MD482 : UDINT;
    MD483 : UDINT;
    MD484 : UDINT;
    MD485 : UDINT;
    MD486 : UDINT;
    MD487 : UDINT;
    MD488 : UDINT;
    MD489 : UDINT;
  END_VAR
  VAR_INPUT
    I : UINT := 0;  (* Индекс фазы *)
    PHASE : TPhaseO;  (* Объект "Вых. фаза" *)
  END_VAR
  VAR
    DIST : DistPhaseO;
  END_VAR

            CASE i OF
0: DIST(PhaseO:=PHASE,MD0=>MD466,MD1=>MD467,MD2=>MD468,MD3=>MD469,MD4=>MD470,MD5=>MD471,MD6=>MD472,MD7=>MD473);
1: DIST(PhaseO:=PHASE,MD0=>MD474,MD1=>MD475,MD2=>MD476,MD3=>MD477,MD4=>MD478,MD5=>MD479,MD6=>MD480,MD7=>MD481);
2: DIST(PhaseO:=PHASE,MD0=>MD482,MD1=>MD483,MD2=>MD484,MD3=>MD485,MD4=>MD486,MD5=>MD487,MD6=>MD488,MD7=>MD489);
END_CASE;

          
END_FUNCTION_BLOCK

(* Запись выходных параметров *)
FUNCTION_BLOCK SetVarO
  VAR_EXTERNAL
    MD460 : UDINT;
    MD461 : UDINT;
    MD462 : UDINT;
    MD463 : UDINT;
    MD464 : UDINT;
    MD465 : UDINT;
  END_VAR
  VAR_INPUT
    VarO : TVarO;  (* Объект "выходные параметры" *)
  END_VAR
  VAR
    DIST : DistVarO;
  END_VAR

            DIST(VarO:=VarO,MD0=>MD460,MD1=>MD461,MD2=>MD462,MD3=>MD463,MD4=>MD464,MD5=>MD465);

          
END_FUNCTION_BLOCK

(* Компоновка состояния элемента *)
FUNCTION m_cond : TCond
  VAR_INPUT
    MD0 : UDINT;
    MD1 : UDINT;
    MD2 : UDINT;
    MD3 : UDINT;
    MD4 : UDINT;
  END_VAR

            m_cond.ID   := UDINT_TO_UINT(MD0/65536);
m_cond.Tmid := UDINT_TO_INT(mod(MD0,65536));

m_cond.Tmin.A[0] := UDINT_TO_INT(MD1/65536);
m_cond.Tmin.A[1] := UDINT_TO_INT(mod(MD1,65536));
m_cond.Tmin.A[2] := UDINT_TO_INT(MD2/65536);
m_cond.Tmin.V    := UDINT_TO_INT(mod(MD2,65536));

m_cond.Tmax.A[0] := UDINT_TO_INT(MD3/65536);
m_cond.Tmax.A[1] := UDINT_TO_INT(mod(MD3,65536));
m_cond.Tmax.A[2] := UDINT_TO_INT(MD4/65536);
m_cond.Tmax.V    := UDINT_TO_INT(mod(MD4,65536));

          
END_FUNCTION

(* Чтение состояния элемента из регистров *)
FUNCTION_BLOCK GetCond
  VAR_EXTERNAL
    MD500 : UDINT;
    MD501 : UDINT;
    MD502 : UDINT;
    MD503 : UDINT;
    MD504 : UDINT;
    MD505 : UDINT;
    MD506 : UDINT;
    MD507 : UDINT;
    MD508 : UDINT;
    MD509 : UDINT;
    MD510 : UDINT;
    MD511 : UDINT;
    MD512 : UDINT;
    MD513 : UDINT;
    MD514 : UDINT;
    MD515 : UDINT;
    MD516 : UDINT;
    MD517 : UDINT;
    MD518 : UDINT;
    MD519 : UDINT;
    MD520 : UDINT;
    MD521 : UDINT;
    MD522 : UDINT;
    MD523 : UDINT;
    MD524 : UDINT;
    MD525 : UDINT;
    MD526 : UDINT;
    MD527 : UDINT;
    MD528 : UDINT;
    MD529 : UDINT;
    MD530 : UDINT;
    MD531 : UDINT;
    MD532 : UDINT;
    MD533 : UDINT;
    MD534 : UDINT;
    MD535 : UDINT;
    MD536 : UDINT;
    MD537 : UDINT;
    MD538 : UDINT;
    MD539 : UDINT;
    MD540 : UDINT;
    MD541 : UDINT;
    MD542 : UDINT;
    MD543 : UDINT;
    MD544 : UDINT;
    MD545 : UDINT;
    MD546 : UDINT;
    MD547 : UDINT;
    MD548 : UDINT;
    MD549 : UDINT;
    MD550 : UDINT;
    MD551 : UDINT;
    MD552 : UDINT;
    MD553 : UDINT;
    MD554 : UDINT;
    MD555 : UDINT;
    MD556 : UDINT;
    MD557 : UDINT;
    MD558 : UDINT;
    MD559 : UDINT;
    MD560 : UDINT;
    MD561 : UDINT;
    MD562 : UDINT;
    MD563 : UDINT;
    MD564 : UDINT;
    MD565 : UDINT;
    MD566 : UDINT;
    MD567 : UDINT;
    MD568 : UDINT;
    MD569 : UDINT;
    MD570 : UDINT;
    MD571 : UDINT;
    MD572 : UDINT;
    MD573 : UDINT;
    MD574 : UDINT;
    MD575 : UDINT;
    MD576 : UDINT;
    MD577 : UDINT;
    MD578 : UDINT;
    MD579 : UDINT;
    MD580 : UDINT;
    MD581 : UDINT;
    MD582 : UDINT;
    MD583 : UDINT;
    MD584 : UDINT;
    MD585 : UDINT;
    MD586 : UDINT;
    MD587 : UDINT;
    MD588 : UDINT;
    MD589 : UDINT;
    MD590 : UDINT;
    MD591 : UDINT;
    MD592 : UDINT;
    MD593 : UDINT;
    MD594 : UDINT;
    MD595 : UDINT;
    MD596 : UDINT;
    MD597 : UDINT;
    MD598 : UDINT;
    MD599 : UDINT;
    MD600 : UDINT;
    MD601 : UDINT;
    MD602 : UDINT;
    MD603 : UDINT;
    MD604 : UDINT;
    MD605 : UDINT;
    MD606 : UDINT;
    MD607 : UDINT;
    MD608 : UDINT;
    MD609 : UDINT;
    MD610 : UDINT;
    MD611 : UDINT;
    MD612 : UDINT;
    MD613 : UDINT;
    MD614 : UDINT;
    MD615 : UDINT;
    MD616 : UDINT;
    MD617 : UDINT;
    MD618 : UDINT;
    MD619 : UDINT;
    MD620 : UDINT;
    MD621 : UDINT;
    MD622 : UDINT;
    MD623 : UDINT;
    MD624 : UDINT;
    MD625 : UDINT;
    MD626 : UDINT;
    MD627 : UDINT;
    MD628 : UDINT;
    MD629 : UDINT;
    MD630 : UDINT;
    MD631 : UDINT;
    MD632 : UDINT;
    MD633 : UDINT;
    MD634 : UDINT;
    MD635 : UDINT;
    MD636 : UDINT;
    MD637 : UDINT;
    MD638 : UDINT;
    MD639 : UDINT;
    MD640 : UDINT;
    MD641 : UDINT;
    MD642 : UDINT;
    MD643 : UDINT;
    MD644 : UDINT;
    MD645 : UDINT;
    MD646 : UDINT;
    MD647 : UDINT;
    MD648 : UDINT;
    MD649 : UDINT;
    MD650 : UDINT;
    MD651 : UDINT;
    MD652 : UDINT;
    MD653 : UDINT;
    MD654 : UDINT;
    MD655 : UDINT;
    MD656 : UDINT;
    MD657 : UDINT;
    MD658 : UDINT;
    MD659 : UDINT;
    MD660 : UDINT;
    MD661 : UDINT;
    MD662 : UDINT;
    MD663 : UDINT;
    MD664 : UDINT;
    MD665 : UDINT;
    MD666 : UDINT;
    MD667 : UDINT;
    MD668 : UDINT;
    MD669 : UDINT;
    MD670 : UDINT;
    MD671 : UDINT;
    MD672 : UDINT;
    MD673 : UDINT;
    MD674 : UDINT;
    MD675 : UDINT;
    MD676 : UDINT;
    MD677 : UDINT;
    MD678 : UDINT;
    MD679 : UDINT;
    MD680 : UDINT;
    MD681 : UDINT;
    MD682 : UDINT;
    MD683 : UDINT;
    MD684 : UDINT;
    MD685 : UDINT;
    MD686 : UDINT;
    MD687 : UDINT;
    MD688 : UDINT;
    MD689 : UDINT;
    MD690 : UDINT;
    MD691 : UDINT;
    MD692 : UDINT;
    MD693 : UDINT;
    MD694 : UDINT;
    MD695 : UDINT;
    MD696 : UDINT;
    MD697 : UDINT;
    MD698 : UDINT;
    MD699 : UDINT;
    MD700 : UDINT;
    MD701 : UDINT;
    MD702 : UDINT;
    MD703 : UDINT;
    MD704 : UDINT;
    MD705 : UDINT;
    MD706 : UDINT;
    MD707 : UDINT;
    MD708 : UDINT;
    MD709 : UDINT;
    MD710 : UDINT;
    MD711 : UDINT;
    MD712 : UDINT;
    MD713 : UDINT;
    MD714 : UDINT;
    MD715 : UDINT;
    MD716 : UDINT;
    MD717 : UDINT;
    MD718 : UDINT;
    MD719 : UDINT;
    MD720 : UDINT;
    MD721 : UDINT;
    MD722 : UDINT;
    MD723 : UDINT;
    MD724 : UDINT;
    MD725 : UDINT;
    MD726 : UDINT;
    MD727 : UDINT;
    MD728 : UDINT;
    MD729 : UDINT;
    MD730 : UDINT;
    MD731 : UDINT;
    MD732 : UDINT;
    MD733 : UDINT;
    MD734 : UDINT;
    MD735 : UDINT;
    MD736 : UDINT;
    MD737 : UDINT;
    MD738 : UDINT;
    MD739 : UDINT;
    MD740 : UDINT;
    MD741 : UDINT;
    MD742 : UDINT;
    MD743 : UDINT;
    MD744 : UDINT;
    MD745 : UDINT;
    MD746 : UDINT;
    MD747 : UDINT;
    MD748 : UDINT;
    MD749 : UDINT;
    MD750 : UDINT;
    MD751 : UDINT;
    MD752 : UDINT;
    MD753 : UDINT;
    MD754 : UDINT;
    MD755 : UDINT;
    MD756 : UDINT;
    MD757 : UDINT;
    MD758 : UDINT;
    MD759 : UDINT;
    MD760 : UDINT;
    MD761 : UDINT;
    MD762 : UDINT;
    MD763 : UDINT;
    MD764 : UDINT;
    MD765 : UDINT;
    MD766 : UDINT;
    MD767 : UDINT;
    MD768 : UDINT;
    MD769 : UDINT;
    MD770 : UDINT;
    MD771 : UDINT;
    MD772 : UDINT;
    MD773 : UDINT;
    MD774 : UDINT;
    MD775 : UDINT;
    MD776 : UDINT;
    MD777 : UDINT;
    MD778 : UDINT;
    MD779 : UDINT;
    MD780 : UDINT;
    MD781 : UDINT;
    MD782 : UDINT;
    MD783 : UDINT;
    MD784 : UDINT;
    MD785 : UDINT;
    MD786 : UDINT;
    MD787 : UDINT;
    MD788 : UDINT;
    MD789 : UDINT;
    MD790 : UDINT;
    MD791 : UDINT;
    MD792 : UDINT;
    MD793 : UDINT;
    MD794 : UDINT;
    MD795 : UDINT;
    MD796 : UDINT;
    MD797 : UDINT;
    MD798 : UDINT;
    MD799 : UDINT;
    MD800 : UDINT;
    MD801 : UDINT;
    MD802 : UDINT;
    MD803 : UDINT;
    MD804 : UDINT;
    MD805 : UDINT;
    MD806 : UDINT;
    MD807 : UDINT;
    MD808 : UDINT;
    MD809 : UDINT;
    MD810 : UDINT;
    MD811 : UDINT;
    MD812 : UDINT;
    MD813 : UDINT;
    MD814 : UDINT;
    MD815 : UDINT;
    MD816 : UDINT;
    MD817 : UDINT;
    MD818 : UDINT;
    MD819 : UDINT;
    MD820 : UDINT;
    MD821 : UDINT;
    MD822 : UDINT;
    MD823 : UDINT;
    MD824 : UDINT;
    MD825 : UDINT;
    MD826 : UDINT;
    MD827 : UDINT;
    MD828 : UDINT;
    MD829 : UDINT;
    MD830 : UDINT;
    MD831 : UDINT;
    MD832 : UDINT;
    MD833 : UDINT;
    MD834 : UDINT;
    MD835 : UDINT;
    MD836 : UDINT;
    MD837 : UDINT;
    MD838 : UDINT;
    MD839 : UDINT;
    MD840 : UDINT;
    MD841 : UDINT;
    MD842 : UDINT;
    MD843 : UDINT;
    MD844 : UDINT;
    MD845 : UDINT;
    MD846 : UDINT;
    MD847 : UDINT;
    MD848 : UDINT;
    MD849 : UDINT;
    MD850 : UDINT;
    MD851 : UDINT;
    MD852 : UDINT;
    MD853 : UDINT;
    MD854 : UDINT;
    MD855 : UDINT;
    MD856 : UDINT;
    MD857 : UDINT;
    MD858 : UDINT;
    MD859 : UDINT;
    MD860 : UDINT;
    MD861 : UDINT;
    MD862 : UDINT;
    MD863 : UDINT;
    MD864 : UDINT;
    MD865 : UDINT;
    MD866 : UDINT;
    MD867 : UDINT;
    MD868 : UDINT;
    MD869 : UDINT;
    MD870 : UDINT;
    MD871 : UDINT;
    MD872 : UDINT;
    MD873 : UDINT;
    MD874 : UDINT;
    MD875 : UDINT;
    MD876 : UDINT;
    MD877 : UDINT;
    MD878 : UDINT;
    MD879 : UDINT;
    MD880 : UDINT;
    MD881 : UDINT;
    MD882 : UDINT;
    MD883 : UDINT;
    MD884 : UDINT;
    MD885 : UDINT;
    MD886 : UDINT;
    MD887 : UDINT;
    MD888 : UDINT;
    MD889 : UDINT;
    MD890 : UDINT;
    MD891 : UDINT;
    MD892 : UDINT;
    MD893 : UDINT;
    MD894 : UDINT;
    MD895 : UDINT;
    MD896 : UDINT;
    MD897 : UDINT;
    MD898 : UDINT;
    MD899 : UDINT;
    MD900 : UDINT;
    MD901 : UDINT;
    MD902 : UDINT;
    MD903 : UDINT;
    MD904 : UDINT;
    MD905 : UDINT;
    MD906 : UDINT;
    MD907 : UDINT;
    MD908 : UDINT;
    MD909 : UDINT;
    MD910 : UDINT;
    MD911 : UDINT;
    MD912 : UDINT;
    MD913 : UDINT;
    MD914 : UDINT;
    MD915 : UDINT;
    MD916 : UDINT;
    MD917 : UDINT;
    MD918 : UDINT;
    MD919 : UDINT;
    MD920 : UDINT;
    MD921 : UDINT;
    MD922 : UDINT;
    MD923 : UDINT;
    MD924 : UDINT;
    MD925 : UDINT;
    MD926 : UDINT;
    MD927 : UDINT;
    MD928 : UDINT;
    MD929 : UDINT;
    MD930 : UDINT;
    MD931 : UDINT;
    MD932 : UDINT;
    MD933 : UDINT;
    MD934 : UDINT;
    MD935 : UDINT;
    MD936 : UDINT;
    MD937 : UDINT;
    MD938 : UDINT;
    MD939 : UDINT;
    MD940 : UDINT;
    MD941 : UDINT;
    MD942 : UDINT;
    MD943 : UDINT;
    MD944 : UDINT;
    MD945 : UDINT;
    MD946 : UDINT;
    MD947 : UDINT;
    MD948 : UDINT;
    MD949 : UDINT;
    MD950 : UDINT;
    MD951 : UDINT;
    MD952 : UDINT;
    MD953 : UDINT;
    MD954 : UDINT;
    MD955 : UDINT;
    MD956 : UDINT;
    MD957 : UDINT;
    MD958 : UDINT;
    MD959 : UDINT;
    MD960 : UDINT;
    MD961 : UDINT;
    MD962 : UDINT;
    MD963 : UDINT;
    MD964 : UDINT;
    MD965 : UDINT;
    MD966 : UDINT;
    MD967 : UDINT;
    MD968 : UDINT;
    MD969 : UDINT;
    MD970 : UDINT;
    MD971 : UDINT;
    MD972 : UDINT;
    MD973 : UDINT;
    MD974 : UDINT;
    MD975 : UDINT;
    MD976 : UDINT;
    MD977 : UDINT;
    MD978 : UDINT;
    MD979 : UDINT;
    MD980 : UDINT;
    MD981 : UDINT;
    MD982 : UDINT;
    MD983 : UDINT;
    MD984 : UDINT;
    MD985 : UDINT;
    MD986 : UDINT;
    MD987 : UDINT;
    MD988 : UDINT;
    MD989 : UDINT;
    MD990 : UDINT;
    MD991 : UDINT;
    MD992 : UDINT;
    MD993 : UDINT;
    MD994 : UDINT;
    MD995 : UDINT;
    MD996 : UDINT;
    MD997 : UDINT;
    MD998 : UDINT;
    MD999 : UDINT;
  END_VAR
  VAR_INPUT
    I : UINT := 0;
  END_VAR
  VAR_OUTPUT
    COND : TCond;
  END_VAR

            CASE i OF
0  : COND := m_cond(MD500,MD501,MD502,MD503,MD504);
1  : COND := m_cond(MD505,MD506,MD507,MD508,MD509);
2  : COND := m_cond(MD510,MD511,MD512,MD513,MD514);
3  : COND := m_cond(MD515,MD516,MD517,MD518,MD519);
4  : COND := m_cond(MD520,MD521,MD522,MD523,MD524);
5  : COND := m_cond(MD525,MD526,MD527,MD528,MD529);
6  : COND := m_cond(MD530,MD531,MD532,MD533,MD534);
7  : COND := m_cond(MD535,MD536,MD537,MD538,MD539);
8  : COND := m_cond(MD540,MD541,MD542,MD543,MD544);
9  : COND := m_cond(MD545,MD546,MD547,MD548,MD549);

10 : COND := m_cond(MD550,MD551,MD552,MD553,MD554);
11 : COND := m_cond(MD555,MD556,MD557,MD558,MD559);
12 : COND := m_cond(MD560,MD561,MD562,MD563,MD564);
13 : COND := m_cond(MD565,MD566,MD567,MD568,MD569);
14 : COND := m_cond(MD570,MD571,MD572,MD573,MD574);
15 : COND := m_cond(MD575,MD576,MD577,MD578,MD579);
16 : COND := m_cond(MD580,MD581,MD582,MD583,MD584);
17 : COND := m_cond(MD585,MD586,MD587,MD588,MD589);
18 : COND := m_cond(MD590,MD591,MD592,MD593,MD594);
19 : COND := m_cond(MD595,MD596,MD597,MD598,MD599);

20 : COND := m_cond(MD600,MD601,MD602,MD603,MD604);
21 : COND := m_cond(MD605,MD606,MD607,MD608,MD609);
22 : COND := m_cond(MD610,MD611,MD612,MD613,MD614);
23 : COND := m_cond(MD615,MD616,MD617,MD618,MD619);
24 : COND := m_cond(MD620,MD621,MD622,MD623,MD624);
25 : COND := m_cond(MD625,MD626,MD627,MD628,MD629);
26 : COND := m_cond(MD630,MD631,MD632,MD633,MD634);
27 : COND := m_cond(MD635,MD636,MD637,MD638,MD639);
28 : COND := m_cond(MD640,MD641,MD642,MD643,MD644);
29 : COND := m_cond(MD645,MD646,MD647,MD648,MD649);

30 : COND := m_cond(MD650,MD651,MD652,MD653,MD654);
31 : COND := m_cond(MD655,MD656,MD657,MD658,MD659);
32 : COND := m_cond(MD660,MD661,MD662,MD663,MD664);
33 : COND := m_cond(MD665,MD666,MD667,MD668,MD669);
34 : COND := m_cond(MD670,MD671,MD672,MD673,MD674);
35 : COND := m_cond(MD675,MD676,MD677,MD678,MD679);
36 : COND := m_cond(MD680,MD681,MD682,MD683,MD684);
37 : COND := m_cond(MD685,MD686,MD687,MD688,MD689);
38 : COND := m_cond(MD690,MD691,MD692,MD693,MD694);
39 : COND := m_cond(MD695,MD696,MD697,MD698,MD699);

40 : COND := m_cond(MD700,MD701,MD702,MD703,MD704);
41 : COND := m_cond(MD705,MD706,MD707,MD708,MD709);
42 : COND := m_cond(MD710,MD711,MD712,MD713,MD714);
43 : COND := m_cond(MD715,MD716,MD717,MD718,MD719);
44 : COND := m_cond(MD720,MD721,MD722,MD723,MD724);
45 : COND := m_cond(MD725,MD726,MD727,MD728,MD729);
46 : COND := m_cond(MD730,MD731,MD732,MD733,MD734);
47 : COND := m_cond(MD735,MD736,MD737,MD738,MD739);
48 : COND := m_cond(MD740,MD741,MD742,MD743,MD744);
49 : COND := m_cond(MD745,MD746,MD747,MD748,MD749);

50 : COND := m_cond(MD750,MD751,MD752,MD753,MD754);
51 : COND := m_cond(MD755,MD756,MD757,MD758,MD759);
52 : COND := m_cond(MD760,MD761,MD762,MD763,MD764);
53 : COND := m_cond(MD765,MD766,MD767,MD768,MD769);
54 : COND := m_cond(MD770,MD771,MD772,MD773,MD774);
55 : COND := m_cond(MD775,MD776,MD777,MD778,MD779);
56 : COND := m_cond(MD780,MD781,MD782,MD783,MD784);
57 : COND := m_cond(MD785,MD786,MD787,MD788,MD789);
58 : COND := m_cond(MD790,MD791,MD792,MD793,MD794);
59 : COND := m_cond(MD795,MD796,MD797,MD798,MD799);

60 : COND := m_cond(MD800,MD801,MD802,MD803,MD804);
61 : COND := m_cond(MD805,MD806,MD807,MD808,MD809);
62 : COND := m_cond(MD810,MD811,MD812,MD813,MD814);
63 : COND := m_cond(MD815,MD816,MD817,MD818,MD819);
64 : COND := m_cond(MD820,MD821,MD822,MD823,MD824);
65 : COND := m_cond(MD825,MD826,MD827,MD828,MD829);
66 : COND := m_cond(MD830,MD831,MD832,MD833,MD834);
67 : COND := m_cond(MD835,MD836,MD837,MD838,MD839);
68 : COND := m_cond(MD840,MD841,MD842,MD843,MD844);
69 : COND := m_cond(MD845,MD846,MD847,MD848,MD849);

70 : COND := m_cond(MD850,MD851,MD852,MD853,MD854);
71 : COND := m_cond(MD855,MD856,MD857,MD858,MD859);
72 : COND := m_cond(MD860,MD861,MD862,MD863,MD864);
73 : COND := m_cond(MD865,MD866,MD867,MD868,MD869);
74 : COND := m_cond(MD870,MD871,MD872,MD873,MD874);
75 : COND := m_cond(MD875,MD876,MD877,MD878,MD879);
76 : COND := m_cond(MD880,MD881,MD882,MD883,MD884);
77 : COND := m_cond(MD885,MD886,MD887,MD888,MD889);
78 : COND := m_cond(MD890,MD891,MD892,MD893,MD894);
79 : COND := m_cond(MD895,MD896,MD897,MD898,MD899);

80 : COND := m_cond(MD900,MD901,MD902,MD903,MD904);
81 : COND := m_cond(MD905,MD906,MD907,MD908,MD909);
82 : COND := m_cond(MD910,MD911,MD912,MD913,MD914);
83 : COND := m_cond(MD915,MD916,MD917,MD918,MD919);
84 : COND := m_cond(MD920,MD921,MD922,MD923,MD924);
85 : COND := m_cond(MD925,MD926,MD927,MD928,MD929);
86 : COND := m_cond(MD930,MD931,MD932,MD933,MD934);
87 : COND := m_cond(MD935,MD936,MD937,MD938,MD939);
88 : COND := m_cond(MD940,MD941,MD942,MD943,MD944);
89 : COND := m_cond(MD945,MD946,MD947,MD948,MD949);

90 : COND := m_cond(MD950,MD951,MD952,MD953,MD954);
91 : COND := m_cond(MD955,MD956,MD957,MD958,MD959);
92 : COND := m_cond(MD960,MD961,MD962,MD963,MD964);
93 : COND := m_cond(MD965,MD966,MD967,MD968,MD969);
94 : COND := m_cond(MD970,MD971,MD972,MD973,MD974);
95 : COND := m_cond(MD975,MD976,MD977,MD978,MD979);
96 : COND := m_cond(MD980,MD981,MD982,MD983,MD984);
97 : COND := m_cond(MD985,MD986,MD987,MD988,MD989);
98 : COND := m_cond(MD990,MD991,MD992,MD993,MD994);
99 : COND := m_cond(MD995,MD996,MD997,MD998,MD999);

END_CASE;
          
END_FUNCTION_BLOCK

(* Компоновка заголовка результатов *)
FUNCTION m_res : TRes
  VAR_INPUT
    MD0 : UDINT;
    MD1 : UDINT;
    MD2 : UDINT;
    MD3 : UDINT;
    MD4 : UDINT;
    MD5 : UDINT;
    MD6 : UDINT;
    MD7 : UDINT;
    MD8 : UDINT;
    MD9 : UDINT;
  END_VAR

            m_res.DR := MD0;  (* секунд от 01-01-1970 *)
m_res.TR := UDINT_TO_TIME(MD1);
m_res.FP := UDINT_TO_TIME(MD2);
m_res.ER := UDINT_TO_UINT(MD3/65536);
m_res.FL := UDINT_TO_WORD(mod(MD3,65536));
m_res.RV[0] := MD4;
m_res.RV[1] := MD5;
m_res.RV[2] := MD6;
m_res.RV[3] := MD7;
m_res.RV[4] := MD8;
m_res.RV[5] := MD9;

          
END_FUNCTION

(* Чтение заголовка результата *)
FUNCTION_BLOCK GetRes
  VAR_EXTERNAL
    MD490 : UDINT;
    MD491 : UDINT;
    MD492 : UDINT;
    MD493 : UDINT;
    MD494 : UDINT;
    MD495 : UDINT;
    MD496 : UDINT;
    MD497 : UDINT;
    MD498 : UDINT;
    MD499 : UDINT;
  END_VAR
  VAR_OUTPUT
    RES : TRes;  (* Объект "заголовок результата" *)
  END_VAR

            RES := m_res(MD490,MD491,MD492,MD493,MD494,MD495,MD496,MD497,MD498,MD499);

          
END_FUNCTION_BLOCK

(* Компоновка Вых. фазы *)
FUNCTION m_phase_out : TPhaseO
  VAR_INPUT
    MD0 : UDINT;
    MD1 : UDINT;
    MD2 : UDINT;
    MD3 : UDINT;
    MD4 : UDINT;
    MD5 : UDINT;
    MD6 : UDINT;
    MD7 : UDINT;
  END_VAR

            m_phase_out.Q0   := UDINT_TO_REAL(MD0);
m_phase_out.Q1   := UDINT_TO_REAL(MD1);
m_phase_out.Q2   := UDINT_TO_REAL(MD2);
m_phase_out.Tin  := UDINT_TO_REAL(MD3);
m_phase_out.Tout := UDINT_TO_REAL(MD4);
m_phase_out.Qm   := UDINT_TO_REAL(MD5);
m_phase_out.Se   := UDINT_TO_REAL(MD6);
m_phase_out.Ve   := UDINT_TO_REAL(MD7);

          
END_FUNCTION

(* Чтение Вых.фазы из регистров *)
FUNCTION_BLOCK GetPhaseO
  VAR_EXTERNAL
    MD466 : UDINT;
    MD467 : UDINT;
    MD468 : UDINT;
    MD469 : UDINT;
    MD470 : UDINT;
    MD471 : UDINT;
    MD472 : UDINT;
    MD473 : UDINT;
    MD474 : UDINT;
    MD475 : UDINT;
    MD476 : UDINT;
    MD477 : UDINT;
    MD478 : UDINT;
    MD479 : UDINT;
    MD480 : UDINT;
    MD481 : UDINT;
    MD482 : UDINT;
    MD483 : UDINT;
    MD484 : UDINT;
    MD485 : UDINT;
    MD486 : UDINT;
    MD487 : UDINT;
    MD488 : UDINT;
    MD489 : UDINT;
  END_VAR
  VAR_INPUT
    I : SINT := 0;  (* Индекс фазы *)
  END_VAR
  VAR_OUTPUT
    PHASE : TPhaseO;  (* Объект "Вых.Фаза" *)
  END_VAR

            CASE i OF
0 : PHASE := m_phase_out(MD466,MD467,MD468,MD469,MD470,MD471,MD472,MD473);
1 : PHASE := m_phase_out(MD474,MD475,MD476,MD477,MD478,MD479,MD480,MD481);
2 : PHASE := m_phase_out(MD482,MD483,MD484,MD485,MD486,MD487,MD488,MD489);
END_CASE;
          
END_FUNCTION_BLOCK

(* Компоновка выходных параметоров *)
FUNCTION m_var_out : TVarO
  VAR_INPUT
    MD0 : UDINT;
    MD1 : UDINT;
    MD2 : UDINT;
    MD3 : UDINT;
    MD4 : UDINT;
    MD5 : UDINT;
  END_VAR

            m_var_out.DTO := MD0;  (* секунд от 01-01-1970 *)
m_var_out.TMO := UDINT_TO_TIME(MD1);
m_var_out.QTY := UDINT_TO_REAL(MD2);
m_var_out.QTS := UDINT_TO_REAL(MD3);
m_var_out.RO1 := UDINT_TO_REAL(MD4);
m_var_out.RO2 := UDINT_TO_REAL(MD5);

          
END_FUNCTION

(* Чтение выходных параметров *)
FUNCTION_BLOCK GetVarO
  VAR_EXTERNAL
    MD460 : UDINT;
    MD461 : UDINT;
    MD462 : UDINT;
    MD463 : UDINT;
    MD464 : UDINT;
    MD465 : UDINT;
  END_VAR
  VAR_OUTPUT
    VarO : TVarO;  (* Объект "выходные параметры" *)
  END_VAR

            VarO := m_var_out(MD460,MD461,MD462,MD463,MD464,MD465);

          
END_FUNCTION_BLOCK

(* Компоновка Вх. фазы *)
FUNCTION m_phase_in : TPhaseI
  VAR_INPUT
    MD0 : UDINT;
    MD1 : UDINT;
    MD2 : UDINT;
    MD3 : UDINT;
    MD4 : UDINT;
    MD5 : UDINT;
    MD6 : UDINT;
    MD7 : UDINT;
  END_VAR

            m_phase_in.Ic   := UDINT_TO_REAL(MD0);
m_phase_in.Tin  := UDINT_TO_REAL(MD1);
m_phase_in.Tout := UDINT_TO_REAL(MD2);
m_phase_in.RN   := UDINT_TO_DWORD(MD3);

m_phase_in.RD[0].A := UINT_TO_SINT(UDINT_TO_UINT(MD4/65536)/256);
m_phase_in.RD[0].B := UINT_TO_SINT(mod(UDINT_TO_UINT(MD4/65536),256));
m_phase_in.RD[1].A := UINT_TO_SINT(UDINT_TO_UINT(mod(MD4,65536))/256);
m_phase_in.RD[1].B := UINT_TO_SINT(mod(UDINT_TO_UINT(mod(MD4,65536)),256));

m_phase_in.RD[2].A := UINT_TO_SINT(UDINT_TO_UINT(MD5/65536)/256);
m_phase_in.RD[2].B := UINT_TO_SINT(mod(UDINT_TO_UINT(MD5/65536),256));
m_phase_in.RD[3].A := UINT_TO_SINT(UDINT_TO_UINT(mod(MD5,65536))/256);
m_phase_in.RD[3].B := UINT_TO_SINT(mod(UDINT_TO_UINT(mod(MD5,65536)),256));

m_phase_in.RD[4].A := UINT_TO_SINT(UDINT_TO_UINT(MD6/65536)/256);
m_phase_in.RD[4].B := UINT_TO_SINT(mod(UDINT_TO_UINT(MD6/65536),256));
m_phase_in.RD[5].A := UINT_TO_SINT(UDINT_TO_UINT(mod(MD6,65536))/256);
m_phase_in.RD[5].B := UINT_TO_SINT(mod(UDINT_TO_UINT(mod(MD6,65536)),256));

m_phase_in.RD[6].A := UINT_TO_SINT(UDINT_TO_UINT(MD7/65536)/256);
m_phase_in.RD[6].B := UINT_TO_SINT(mod(UDINT_TO_UINT(MD7/65536),256));
m_phase_in.RD[7].A := UINT_TO_SINT(UDINT_TO_UINT(mod(MD7,65536))/256);
m_phase_in.RD[7].B := UINT_TO_SINT(mod(UDINT_TO_UINT(mod(MD7,65536)),256));

          
END_FUNCTION

(* Чтение Вх.фазы из регистров *)
FUNCTION_BLOCK GetPhaseI
  VAR_EXTERNAL
    MD436 : UDINT;
    MD437 : UDINT;
    MD438 : UDINT;
    MD439 : UDINT;
    MD440 : UDINT;
    MD441 : UDINT;
    MD442 : UDINT;
    MD443 : UDINT;
    MD444 : UDINT;
    MD445 : UDINT;
    MD446 : UDINT;
    MD447 : UDINT;
    MD448 : UDINT;
    MD449 : UDINT;
    MD450 : UDINT;
    MD451 : UDINT;
    MD452 : UDINT;
    MD453 : UDINT;
    MD454 : UDINT;
    MD455 : UDINT;
    MD456 : UDINT;
    MD457 : UDINT;
    MD458 : UDINT;
    MD459 : UDINT;
  END_VAR
  VAR_INPUT
    I : SINT := 0;  (* Индекс фазы *)
  END_VAR
  VAR_OUTPUT
    PHASE : TPhaseI;  (* Объект "Вх.фаза" *)
  END_VAR

            CASE i OF
0 : PHASE := m_phase_in(MD436,MD437,MD438,MD439,MD440,MD441,MD442,MD443);
1 : PHASE := m_phase_in(MD444,MD445,MD446,MD447,MD448,MD449,MD450,MD451);
2 : PHASE := m_phase_in(MD452,MD453,MD454,MD455,MD456,MD457,MD458,MD459);
END_CASE;
          
END_FUNCTION_BLOCK

(* Компоновка входных параметоров *)
FUNCTION m_var_in : TVarI
  VAR_INPUT
    MD0 : UDINT;
    MD1 : UDINT;
    MD2 : UDINT;
    MD3 : UDINT;
    MD4 : UDINT;
    MD5 : UDINT;
  END_VAR

            m_var_in.DTI := MD0; (* секунд от 01-01-1970 *)
m_var_in.TMI := UDINT_TO_TIME(MD1);
m_var_in.TOV := UDINT_TO_REAL(MD2);
m_var_in.MHT := UDINT_TO_REAL(MD3);
m_var_in.RI1 := UDINT_TO_REAL(MD4);
m_var_in.RI2 := UDINT_TO_REAL(MD5);

          
END_FUNCTION

(* Чтение входных параметров *)
FUNCTION_BLOCK GetVarI
  VAR_EXTERNAL
    MD430 : UDINT;
    MD431 : UDINT;
    MD432 : UDINT;
    MD433 : UDINT;
    MD434 : UDINT;
    MD435 : UDINT;
  END_VAR
  VAR_OUTPUT
    VarI : TVarI;  (* Объект "входные параметры" *)
  END_VAR

            VarI := m_var_in(MD430,MD431,MD432,MD433,MD434,MD435);

          
END_FUNCTION_BLOCK

(* Компоновка радиатора *)
FUNCTION m_rad : TRad
  VAR_INPUT
    MD0 : UDINT;
    MD1 : UDINT;
    MD2 : UDINT;
    MD3 : UDINT;
    MD4 : UDINT;
    MD5 : UDINT;
    MD6 : UDINT;
    MD7 : UDINT;
  END_VAR

            m_rad.Vm := UDINT_TO_REAL(MD0);
m_rad.Fk := UDINT_TO_REAL(MD1);
m_rad.Q0 := UDINT_TO_REAL(MD2);
m_rad.Q1 := UDINT_TO_REAL(MD3);
m_rad.BL[0] := UDINT_TO_REAL(MD4);
m_rad.BL[1] := UDINT_TO_REAL(MD5);
m_rad.BL[2] := UDINT_TO_REAL(MD6);
m_rad.BL[3] := UDINT_TO_REAL(MD7);

          
END_FUNCTION

(* Чтение радиатора из регистров *)
FUNCTION_BLOCK GetRad
  VAR_EXTERNAL
    MD302 : UDINT;
    MD303 : UDINT;
    MD304 : UDINT;
    MD305 : UDINT;
    MD306 : UDINT;
    MD307 : UDINT;
    MD308 : UDINT;
    MD309 : UDINT;
    MD310 : UDINT;
    MD311 : UDINT;
    MD312 : UDINT;
    MD313 : UDINT;
    MD314 : UDINT;
    MD315 : UDINT;
    MD316 : UDINT;
    MD317 : UDINT;
    MD318 : UDINT;
    MD319 : UDINT;
    MD320 : UDINT;
    MD321 : UDINT;
    MD322 : UDINT;
    MD323 : UDINT;
    MD324 : UDINT;
    MD325 : UDINT;
    MD326 : UDINT;
    MD327 : UDINT;
    MD328 : UDINT;
    MD329 : UDINT;
    MD330 : UDINT;
    MD331 : UDINT;
    MD332 : UDINT;
    MD333 : UDINT;
    MD334 : UDINT;
    MD335 : UDINT;
    MD336 : UDINT;
    MD337 : UDINT;
    MD338 : UDINT;
    MD339 : UDINT;
    MD340 : UDINT;
    MD341 : UDINT;
    MD342 : UDINT;
    MD343 : UDINT;
    MD344 : UDINT;
    MD345 : UDINT;
    MD346 : UDINT;
    MD347 : UDINT;
    MD348 : UDINT;
    MD349 : UDINT;
    MD350 : UDINT;
    MD351 : UDINT;
    MD352 : UDINT;
    MD353 : UDINT;
    MD354 : UDINT;
    MD355 : UDINT;
    MD356 : UDINT;
    MD357 : UDINT;
    MD358 : UDINT;
    MD359 : UDINT;
    MD360 : UDINT;
    MD361 : UDINT;
    MD362 : UDINT;
    MD363 : UDINT;
    MD364 : UDINT;
    MD365 : UDINT;
    MD366 : UDINT;
    MD367 : UDINT;
    MD368 : UDINT;
    MD369 : UDINT;
    MD370 : UDINT;
    MD371 : UDINT;
    MD372 : UDINT;
    MD373 : UDINT;
    MD374 : UDINT;
    MD375 : UDINT;
    MD376 : UDINT;
    MD377 : UDINT;
    MD378 : UDINT;
    MD379 : UDINT;
    MD380 : UDINT;
    MD381 : UDINT;
    MD382 : UDINT;
    MD383 : UDINT;
    MD384 : UDINT;
    MD385 : UDINT;
    MD386 : UDINT;
    MD387 : UDINT;
    MD388 : UDINT;
    MD389 : UDINT;
    MD390 : UDINT;
    MD391 : UDINT;
    MD392 : UDINT;
    MD393 : UDINT;
    MD394 : UDINT;
    MD395 : UDINT;
    MD396 : UDINT;
    MD397 : UDINT;
    MD398 : UDINT;
    MD399 : UDINT;
    MD400 : UDINT;
    MD401 : UDINT;
    MD402 : UDINT;
    MD403 : UDINT;
    MD404 : UDINT;
    MD405 : UDINT;
    MD406 : UDINT;
    MD407 : UDINT;
    MD408 : UDINT;
    MD409 : UDINT;
    MD410 : UDINT;
    MD411 : UDINT;
    MD412 : UDINT;
    MD413 : UDINT;
    MD414 : UDINT;
    MD415 : UDINT;
    MD416 : UDINT;
    MD417 : UDINT;
    MD418 : UDINT;
    MD419 : UDINT;
    MD420 : UDINT;
    MD421 : UDINT;
    MD422 : UDINT;
    MD423 : UDINT;
    MD424 : UDINT;
    MD425 : UDINT;
    MD426 : UDINT;
    MD427 : UDINT;
    MD428 : UDINT;
    MD429 : UDINT;
  END_VAR
  VAR_INPUT
    I : SINT := 0;  (* Индекс профиля *)
  END_VAR
  VAR_OUTPUT
    RAD : TRad;  (* Объект "профиль" *)
  END_VAR

            CASE i OF
0 : RAD := m_rad(MD302,MD303,MD304,MD305,MD306,MD307,MD308,MD309);
1 : RAD := m_rad(MD310,MD311,MD312,MD313,MD314,MD315,MD316,MD317);
2 : RAD := m_rad(MD318,MD319,MD320,MD321,MD322,MD323,MD324,MD325);
3 : RAD := m_rad(MD326,MD327,MD328,MD329,MD330,MD331,MD332,MD333);
4 : RAD := m_rad(MD334,MD335,MD336,MD337,MD338,MD339,MD340,MD341);
5 : RAD := m_rad(MD342,MD343,MD344,MD345,MD346,MD347,MD348,MD349);
6 : RAD := m_rad(MD350,MD351,MD352,MD353,MD354,MD355,MD356,MD357);
7 : RAD := m_rad(MD358,MD359,MD360,MD361,MD362,MD363,MD364,MD365);
8 : RAD := m_rad(MD366,MD367,MD368,MD369,MD370,MD371,MD372,MD373);
9 : RAD := m_rad(MD374,MD375,MD376,MD377,MD378,MD379,MD380,MD381);
10: RAD := m_rad(MD382,MD383,MD384,MD385,MD386,MD387,MD388,MD389);
11: RAD := m_rad(MD390,MD391,MD392,MD393,MD394,MD395,MD396,MD397);
12: RAD := m_rad(MD398,MD399,MD400,MD401,MD402,MD403,MD404,MD405);
13: RAD := m_rad(MD406,MD407,MD408,MD409,MD410,MD411,MD412,MD413);
14: RAD := m_rad(MD414,MD415,MD416,MD417,MD418,MD419,MD420,MD421);
15: RAD := m_rad(MD422,MD423,MD424,MD425,MD426,MD427,MD428,MD429);
END_CASE;
          
END_FUNCTION_BLOCK

(* Компоновка концигурации объекта *)
FUNCTION m_conf : TConf
  VAR_INPUT
    MD0 : UDINT;
    MD1 : UDINT;
  END_VAR

            m_conf.Nm := UDINT_TO_UINT(MD0/65536);
m_conf.Nr := UDINT_TO_UINT(mod(MD0,65536));
m_conf.Tc := UDINT_TO_TIME(MD1);

          
END_FUNCTION

(* Чтение конфигурации из регистров *)
FUNCTION_BLOCK GetConf
  VAR_EXTERNAL
    MD300 : UDINT;
    MD301 : UDINT;
  END_VAR
  VAR_OUTPUT
    CONF : TConf;  (* Конфигурация объекта *)
  END_VAR

            CONF := m_conf(MD300,MD301);

          
END_FUNCTION_BLOCK

(* Выдает строку по коду ошибки *)
FUNCTION LogErr : STRING
  VAR_INPUT
    ERR : TError := E_SUCCESS;  (* Флаг отладочной печати *)
  END_VAR

            LogErr := LogMsg('',Info,ERR);



          
END_FUNCTION

(* Строка ID в 16# представлении *)
FUNCTION Byte2Str : STRING
  VAR_INPUT
    Bt : BYTE := 0;  (* Входной байт *)
  END_VAR
  VAR
    i : SINT := 0;  (* Индекс бита *)
    str : STRING := '2#';  (* Итоговая строка *)
  END_VAR

            for i:=7 to 0 by -1 do
  if ((Bt and shl(1, i))<>0) then
    str:=MakeMsg(str, '1');
  else
    str:=MakeMsg(str, '0');
  end_if;
end_for;
Byte2Str:=str;

          
END_FUNCTION

FUNCTION REAL2UDI : UDINT
  VAR_INPUT
    VALUE : REAL := 0.0;
  END_VAR
  VAR
    tmp : UDINT := 0;
  END_VAR

            {{
  union { UDINT  udint; float real; } value;
  value.real = VALUE;
  TMP = value.udint;
}}
REAL2UDI := TMP;

          
END_FUNCTION

(* Cвойства масла от температуры *)
FUNCTION mat_oil : TMat
  VAR_INPUT
    Tm : REAL := 20.0;  (* Температура масла *)
  END_VAR

            mat_oil.kt := 0.1124  - 0.000085 * Tm;
mat_oil.pl := 892.0   - 0.6075   * Tm;
mat_oil.cp := 1549.0  + 5.93334  * Tm;
mat_oil.md := 0.13515 * exp(2820.0/(272.0+1.13*Tm))/100000.0;

          
END_FUNCTION

(* Конфигурация модели *)
PROGRAM P_EVAL
  VAR
    LocalVar0 : DINT;
  END_VAR

            LocalVar0:=0;
          
END_PROGRAM

